# EPICS substitutions: ethmodApp/Db/AKI2C_DS28CM00.substitutions
file AKI2C_DS28CM00_dev.template
{
   pattern { P    ,R    ,PORT    ,ADDR     ,TIMEOUT     }
           { $(P) ,$(R) ,$(PORT) ,$(ADDR)  ,$(TIMEOUT)  }
}
